FUNCTION alg_a_ejectpulse : BOOL
VAR_INPUT
	state: STATE;
END_VAR

alg_a_ejectpulse := state.dvar_M_vacuum_a_ejectpulse;

END_FUNCTION

(* stored: Version 1.1.0.1, ProductVersion 3.1.4022.18
   POU alg_a_ejectpulse: Id {1d3eb04b-0a2a-4415-808e-8ab9e178e08e}, SpecialFunc None *)
